// TwinCAT 3 PLC project MainProject
// ProgramVersion: 3.1.4023.0
// libraries:
//   Tc2_Standard, * (Beckhoff Automation GmbH)
//   Tc2_System, * (Beckhoff Automation GmbH)
//   Tc3_Module, * (Beckhoff Automation GmbH)
// project tree:
//   / PlcTask.TcTTO
//   POUs/Devices/ I_Cylinder.TcIO, T_Cylinder.TcPOU
//   POUs/ MAIN.TcPOU, T_LidApplyStation.TcPOU, T_Station.TcPOU
// real-time tasks:
//   TASK PlcTask: cycle T#10ms, priority 20, ADS port 350

CONFIGURATION MainProject
    RESOURCE PLC ON TwinCAT3
        TASK PlcTask(INTERVAL := T#10ms, PRIORITY := 20);
        PROGRAM MAIN WITH PlcTask : MAIN;
    END_RESOURCE
END_CONFIGURATION

// ---- POUs/Devices/I_Cylinder.TcIO
INTERFACE I_Cylinder

METHOD PUBLIC Extend
VAR_INPUT
END_VAR
END_METHOD

METHOD PUBLIC Retract
VAR_INPUT
END_VAR
END_METHOD

END_INTERFACE

// ---- POUs/MAIN.TcPOU
PROGRAM MAIN
VAR
	LidApplicatiorCylinder : T_Cylinder;
	LidApplyStation : T_LidApplyStation(Cylinder := LidApplicatiorCylinder);

	start: BOOL;
END_VAR

LidApplyStation();

IF start THEN
	start := FALSE;
	LidApplyStation.Start();
END_IF

END_PROGRAM

// ---- POUs/Devices/T_Cylinder.TcPOU
FUNCTION_BLOCK T_Cylinder IMPLEMENTS I_Cylinder
VAR_INPUT
END_VAR
VAR_OUTPUT
END_VAR
VAR
	output AT %Q* : BOOL;
END_VAR

METHOD PUBLIC Extend
VAR_INPUT
END_VAR
output := true;
END_METHOD

METHOD PUBLIC Retract
VAR_INPUT
END_VAR
output := false;
END_METHOD

END_FUNCTION_BLOCK

// ---- POUs/T_LidApplyStation.TcPOU
FUNCTION_BLOCK T_LidApplyStation EXTENDS T_Station
VAR_INPUT
END_VAR
VAR_OUTPUT
END_VAR
VAR
	processState : (IDLE,EXTEND_APPLICATOR_ARM, WAIT,RETRACT_APPLICATOR_ARM, COMPLETE);
	waitTimer : TON;
	cylinder : I_Cylinder; 
END_VAR
VAR CONSTANT
	PROCESS_TIME : TIME := T#2S;
END_VAR

super^();

METHOD PROTECTED Execute
VAR_INPUT
END_VAR


CASE processState OF
	
	IDLE : // 
	
		waitTimer(IN:=FALSE);
		processState := EXTEND_APPLICATOR_ARM;
	
	EXTEND_APPLICATOR_ARM : // 
	
		cylinder.Extend();
		processState := WAIT;
	
	WAIT : //
	
		waitTimer(IN:=TRUE, PT:=PROCESS_TIME);
		IF waitTimer.Q THEN
			processState := RETRACT_APPLICATOR_ARM;
		END_IF
	
	RETRACT_APPLICATOR_ARM : //
	
		cylinder.Retract();
		processState := COMPLETE;
	
	COMPLETE: //
	
		StateComplete();
		processState := IDLE;

END_CASE
END_METHOD

METHOD FB_init : BOOL
VAR_INPUT
	bInitRetains : BOOL; // if TRUE, the retain variables are initialized (warm start / cold start)
	bInCopyCode : BOOL;  // if TRUE, the instance afterwards gets moved into the copy code (online change)
	Cylinder : I_Cylinder;
END_VAR
this^.cylinder := Cylinder;
END_METHOD

END_FUNCTION_BLOCK

// ---- POUs/T_Station.TcPOU
FUNCTION_BLOCK T_Station
VAR_INPUT
END_VAR
VAR_OUTPUT
END_VAR
VAR
	StationState : (UNINITIALISED,INITIALISING,IDLE,STARTING,EXECUTE,COMPLETING,COMPLETE,STOPPING,STOPPED,RESETTING,HOLDING,HELD,UNHOLDING,SUSPENDING,SUSPENDED,UNSUSPENDING,CLEARING,ABORTED,ABORTING) := UNINITIALISED;
END_VAR

CASE StationState OF
	
	UNINITIALISED : Uninitialised();
	INITIALISING : Initialising();
	IDLE : Idle();
	STARTING : Starting();
	EXECUTE : Execute();
	COMPLETING : Completing();
	COMPLETE : Complete();
	STOPPING : Stopping();
	STOPPED : Stopped();
	RESETTING : Resetting();
	HOLDING : Holding();
	HELD : Held();
	UNHOLDING : Unholding();
	SUSPENDING : Suspending();
	SUSPENDED : Suspended();
	UNSUSPENDING : Unsuspending();
	CLEARING : Clearing();
	ABORTED : Aborted();
	ABORTING : Aborting();

	
END_CASE

METHOD PUBLIC Abort
VAR_INPUT
END_VAR
StationState := ABORTING;
END_METHOD

METHOD PROTECTED Aborted
VAR_INPUT
END_VAR
Clear();
END_METHOD

METHOD PROTECTED Aborting
VAR_INPUT
END_VAR
StateComplete();
END_METHOD

METHOD PUBLIC Clear
VAR_INPUT
END_VAR
IF StationState = ABORTED THEN 
	StationState := CLEARING;
END_IF
END_METHOD

METHOD PROTECTED Clearing
VAR_INPUT
END_VAR
StateComplete();
END_METHOD

METHOD PROTECTED Complete
VAR_INPUT
END_VAR
Reset();
END_METHOD

METHOD PROTECTED Completing
VAR_INPUT
END_VAR
StateComplete();
END_METHOD

METHOD PROTECTED Execute
VAR_INPUT
END_VAR
StateComplete();
END_METHOD

METHOD PROTECTED Held
VAR_INPUT
END_VAR
Unhold();
END_METHOD

METHOD PUBLIC Hold
VAR_INPUT
END_VAR
IF StationState = EXECUTE THEN 
	StationState := HOLDING;
END_IF
END_METHOD

METHOD PROTECTED Holding
VAR_INPUT
END_VAR
StateComplete();
END_METHOD

METHOD PROTECTED Idle
VAR_INPUT
END_VAR
END_METHOD

METHOD PUBLIC Initialise
VAR_INPUT
END_VAR
IF StationState = UNINITIALISED THEN 
	StationState := INITIALISING;
END_IF
END_METHOD

METHOD PROTECTED Initialising
VAR_INPUT
END_VAR
StateComplete();
END_METHOD

PROPERTY PUBLIC isExecuting : bool
GET
isExecuting := (StationState = EXECUTE);
END_GET
END_PROPERTY

PROPERTY PUBLIC isInitialised : bool
GET
isInitialised := (StationState <> UNINITIALISED);
END_GET
END_PROPERTY

PROPERTY PUBLIC isStopped : BOOL
GET
isStopped := (StationState = STOPPED);
END_GET
END_PROPERTY

METHOD PUBLIC Reset
VAR_INPUT
END_VAR
IF (StationState = STOPPED) or (StationState = COMPLETE) THEN 
	StationState := RESETTING;
END_IF
END_METHOD

METHOD PROTECTED Resetting
VAR_INPUT
END_VAR
StateComplete();
END_METHOD

METHOD PUBLIC Start
VAR_INPUT
END_VAR
IF StationState = IDLE THEN 
	StationState := STARTING;
END_IF
END_METHOD

METHOD PROTECTED Starting
VAR_INPUT
END_VAR
StateComplete();
END_METHOD

METHOD PROTECTED StateComplete
VAR_INPUT
END_VAR
CASE StationState OF 
	
	UNINITIALISED : RETURN;
	INITIALISING : StationState := IDLE;
	IDLE : RETURN;
	STARTING : StationState := EXECUTE;
	EXECUTE : StationState := COMPLETING;
	COMPLETING : StationState := COMPLETE;
	COMPLETE : RETURN;
	STOPPING : StationState := STOPPED;
	STOPPED : RETURN;
	RESETTING : StationState := IDLE;
	HOLDING : StationState := HELD;
	HELD : RETURN;
	UNHOLDING : StationState := EXECUTE;
	SUSPENDING : StationState := SUSPENDED;
	SUSPENDED : RETURN;
	UNSUSPENDING : StationState := EXECUTE;
	CLEARING : StationState := STOPPED;
	ABORTED : RETURN;
	ABORTING : StationState := ABORTED;
	
END_CASE
END_METHOD

METHOD PUBLIC Stop
VAR_INPUT
END_VAR
CASE StationState OF
	STOPPED: RETURN;
	STOPPING: RETURN;
	CLEARING: RETURN;
	ABORTED: RETURN;
	ABORTING: RETURN;
END_CASE

StationState := STOPPING;
END_METHOD

METHOD PROTECTED Stopped
VAR_INPUT
END_VAR
Reset();
END_METHOD

METHOD PROTECTED Stopping
VAR_INPUT
END_VAR
StateComplete();
END_METHOD

METHOD PUBLIC Suspend
VAR_INPUT
END_VAR
IF StationState = EXECUTE THEN 
	StationState := SUSPENDING;
END_IF
END_METHOD

METHOD PROTECTED Suspended
VAR_INPUT
END_VAR
Unsuspended();
END_METHOD

METHOD PROTECTED Suspending
VAR_INPUT
END_VAR
StateComplete();
END_METHOD

METHOD PUBLIC Unhold
VAR_INPUT
END_VAR
IF StationState = HELD THEN 
	StationState := UNHOLDING;
END_IF
END_METHOD

METHOD PROTECTED Unholding
VAR_INPUT
END_VAR
StateComplete();
END_METHOD

METHOD PROTECTED Uninitialised
VAR_INPUT
END_VAR
Initialise();
END_METHOD

METHOD PUBLIC Unsuspended
VAR_INPUT
END_VAR
IF StationState = SUSPENDED THEN 
	StationState := UNSUSPENDING;
END_IF
END_METHOD

METHOD PROTECTED Unsuspending
VAR_INPUT
END_VAR
StateComplete();
END_METHOD

END_FUNCTION_BLOCK
